// TIA Portal V17 export
// export: Created 2024-09-03T21:54:55.8153134Z, ExportSetting WithDefaults, DisplayName Totally Integrated Automation Portal, DisplayVersion V17 Update 7, DisplayName TIA Portal Openness, DisplayVersion V17 Update 7, DisplayName TIA Portal Version Control Interface, DisplayVersion V17, DisplayName SINAMICS Startdrive Advanced, DisplayVersion V17 SP2, DisplayName SINAMICS Startdrive G110M, G120, G120C, G120D, G120P, G115D, DisplayVersion V17 SP2, DisplayName SINAMICS Startdrive G130, G150, S120, S150, SINAMICS MV, S210, DisplayVersion V17 SP2, DisplayName STEP 7 Professional, DisplayVersion V17 Update 7, DisplayName STEP 7 Safety, DisplayVersion V17 Update 6, DisplayName WinCC Advanced / Unified PC, DisplayVersion V17 Update 7
DATA_BLOCK "StationParameters"   // DB9
{ S7_Optimized_Access := 'TRUE' }
VERSION : 0.1
// stored: AutoNumber true, DBAccessibleFromOPCUA true, DBAccessibleFromWebserver true, IsOnlyStoredInLoadMemory false, IsRetainMemResEnabled false, IsWriteProtectedInAS false, MemoryReserve 100
   VAR RETAIN
      PumpStopDelay : Time := T#2S;
      ReleasePressureDelay : Time := T#5S;
      VH1BasicPositionMin : Real := -5.0;
      VH1BasicPositionMax : Real := 10.0;
      VH2BasicPositionMin : Real := -5.0;
      VH2BasicPositionMax : Real := 10.0;
      DisableScanner : Bool := TRUE;
      NOKBoxSize : Int := 3;
      OKUpperStockSize : Int := 3;
      OKLowerStockSize : Int := 3;
      GhostMode : Bool := FALSE;
      VH1MaxPosition : Real := 63.0;
      VH2MaxPosition : Real := 63.0;
      MaximalFittingTime : Time := T#20S;
      DisableR1Detection1 : Bool := FALSE;
      DisableR1Detection2 : Bool := FALSE;
      ManipulatorTimeBeforeLowerFixation : Time := T#5S;
      HangerDetectionORfunction : Bool := FALSE;
      AudioSignalizationTimeBeforeSafety : Time := T#5S;
      Servo : "UDT_ServoPrameters";
      ServoPositions { S7_SetPoint := 'True'} : Array[0..9] of DInt;
      DontUseHangerForParts { S7_SetPoint := 'True'} : Bool := TRUE;
      ManipulatorCommOff { S7_SetPoint := 'True'} : Bool := TRUE;
   END_VAR
BEGIN
   Servo.Velocity := 500;
   Servo.OverV := 100;
   Servo.OverAcc := 50;
   Servo.OverDec := 100;
   ServoPositions[0] := 10002;
   ServoPositions[1] := 784500;
   ServoPositions[2] := 1510500;
   ServoPositions[3..9] := 0;
END_DATA_BLOCK
